// Mitsubishi GX Works2 project: 20150903   PLC: Q03UDV

PROGRAM P1
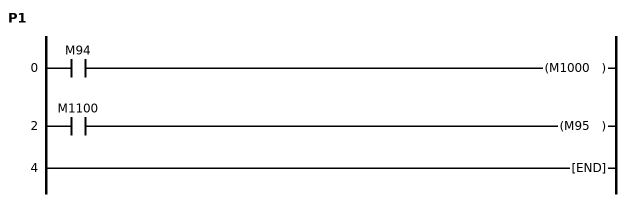
0     LD      M94
      OUT     M1000
2     LD      M1100
      OUT     M95
4     END
END_PROGRAM

PROGRAM P2
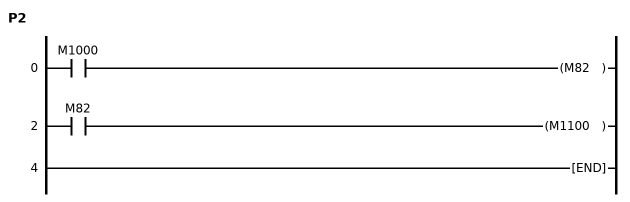
0     LD      M1000
      OUT     M82
2     LD      M82
      OUT     M1100
4     END
END_PROGRAM
